// TIA Portal V20 export
// export: Created 2026-07-16T13:01:16.423654Z, ExportSetting WithDefaults, DisplayName Totally Integrated Automation Portal, DisplayVersion V20 Update 5, DisplayName TIA Portal Openness, DisplayVersion V20 Update 4, DisplayName TIA Portal Version Control Interface, DisplayVersion V20 Update 5, DisplayName SINAMICS Startdrive Advanced, DisplayVersion V20, DisplayName SINAMICS DCC, DisplayVersion V20, DisplayName SINAMICS Startdrive G130, G150, S120, S150, SINAMICS MV, G220, S200, S210, DisplayVersion V20, DisplayName SINAMICS Startdrive G110M, G120, G120C, G120D, G120P, G115D, DisplayVersion V20, DisplayName STEP 7 Professional, DisplayVersion V20 Update 5, DisplayName STEP 7 Safety, DisplayVersion V20 Update 2, DisplayName WinCC Basic/Comfort/Advanced, DisplayVersion V20 Update 5, DisplayName WinCC Unified, DisplayVersion V20 Update 5
VAR_GLOBAL   // PLC tag table "Default tag table"
   Tag_1 AT %I500.0 : Bool;
   Tag_2 AT %I500.1 : Bool;
   Tag_3 AT %I500.2 : Bool;
   Tag_4 AT %I500.3 : Bool;
   Tag_5 AT %I500.6 : Bool;
   Tag_6 AT %I500.7 : Bool;
   Tag_7 AT %I501.0 : Bool;
   Tag_8 AT %I501.1 : Bool;
   Tag_9 AT %I501.2 : Bool;
   Tag_10 AT %I501.3 : Bool;
   Tag_11 AT %I501.4 : Bool;
   Tag_12 AT %I501.5 : Bool;
   Tag_13 AT %I501.6 : Bool;
   Tag_14 AT %I501.7 : Bool;
   Tag_15 AT %I502.1 : Bool;
   Tag_16 AT %I502.2 : Bool;
   Tag_17 AT %I502.3 : Bool;
   Tag_18 AT %I502.4 : Bool;
   Tag_19 AT %I502.5 : Bool;
   Tag_20 AT %I502.6 : Bool;
   Tag_21 AT %I502.7 : Bool;
   Tag_22 AT %I503.0 : Bool;
   Tag_23 AT %I503.1 : Bool;
   Tag_24 AT %I503.2 : Bool;
   Tag_25 AT %I503.3 : Bool;
   Tag_26 AT %I503.4 : Bool;
   Tag_41 AT %IW508 : Word;
   Tag_42 AT %IW528 : Word;
   Tag_43 AT %IW532 : Word;
   Tag_44 AT %IW650 : Word;
   Tag_45 AT %IW64 : Word;
   Tag_46 AT %IW66 : Word;
   Tag_47 AT %IW68 : Word;
   Tag_48 AT %IW70 : Word;
   Tag_49 AT %IW72 : Word;
   Tag_50 AT %IW74 : Word;
   Tag_51 AT %IW76 : Word;
   Tag_52 AT %IW78 : Word;
   Tag_27 AT %Q500.0 : Bool;
   Tag_28 AT %Q500.1 : Bool;
   Tag_29 AT %Q500.2 : Bool;
   Tag_30 AT %Q500.4 : Bool;
   Tag_31 AT %Q500.5 : Bool;
   Tag_32 AT %Q501.0 : Bool;
   Tag_33 AT %Q501.1 : Bool;
   Tag_34 AT %Q501.2 : Bool;
   Tag_35 AT %Q501.3 : Bool;
   Tag_36 AT %Q501.4 : Bool;
   Tag_37 AT %Q501.5 : Bool;
   Tag_38 AT %Q502.0 : Bool;
   Tag_39 AT %Q502.1 : Bool;
   Tag_40 AT %Q502.2 : Bool;
   Tag_53 AT %QW64 : Word;
   Tag_54 AT %QW66 : Word;
   "Clock_0.5Hz" AT %M0.7 : Bool;
   AirStarWord0IN AT %IW80 : Word;
   AirStarWord2IN AT %IW82 : Word;
   AirStarWord0OUT AT %QW68 : Word;
   AirStarWord2OUT AT %QW70 : Word;
   FirstScan AT %M1.0 : Bool;
   AlwaysTrue AT %M1.2 : Bool;
   DI1_SYS_ControlHealthy AT %I0.0 : Bool;   // Safety/control circuit healthy
   DI2_SPR_1 AT %I0.1 : Bool;   // Spare (wired to -X3:1)
   DI3_SYS_CycleStart AT %I0.2 : Bool;   // Cycle start pushbutton (local/remote)
   DI4_SYS_CycleStop AT %I0.3 : Bool;   // Cycle stop pushbutton (NC)
   DI5_SHR_RunFwdFB AT %I0.4 : Bool;   // Shredder running forward feedback
   DI6_SHR_RunRevFB AT %I0.5 : Bool;   // Shredder running reverse feedback
   DI7_SYS_MotorFault AT %I0.6 : Bool;   // Motor fault (soft start fault relay)
   DI8_HPR_LevelHigh AT %I0.7 : Bool;   // Hopper high level sensor
   DI9_IFC_Running AT %I1.0 : Bool;   // Infeed conveyor running feedback
   DI10_DIS_Running AT %I1.1 : Bool;   // Discharge conveyor running feedback
   DI11_PSH_PowerPackRunning AT %I1.2 : Bool;   // Pusher power pack running feedback
   DI12_PSH_HomeLimit AT %I1.3 : Bool;   // Pusher parked/home position
   DI13_PSH_FullTravelLimit AT %I1.4 : Bool;   // Pusher fully extended position
   DI14_PSH_HighPressure AT %I1.5 : Bool;   // Pusher hydraulic high pressure switch
   DI15_SYS_DownstreamRunning AT %I2.0 : Bool;   // Downstream equipment running
   DI16_PSH_LocalRemote AT %I2.1 : Bool;   // Pusher operation local/remote selector
   DI17_SPR_2 AT %I2.2 : Bool;   // Spare (wired to terminal)
   DI18_SPR_3 AT %I2.3 : Bool;   // Spare (wired to terminal)
   DI19_SPR_4 AT %I2.4 : Bool;   // Spare (wired to terminal)
   DI20_SPR_5 AT %I2.5 : Bool;   // Spare (wired to terminal)
   DI21_SPR_6 AT %I2.6 : Bool;   // Spare (wired to terminal)
   DI22_SPR_7 AT %I2.7 : Bool;   // Spare (wired to terminal)
   DQ1_SHR_RunFwd AT %Q0.0 : Bool;   // Run shredder forward command
   DQ2_SHR_RunRev AT %Q0.1 : Bool;   // Run shredder reverse command
   DQ3_PSH_RunPowerPack AT %Q0.2 : Bool;   // Run pusher power pack command
   DQ4_IFC_Run AT %Q0.3 : Bool;   // Run infeed conveyor command
   DQ5_DIS_Run AT %Q0.4 : Bool;   // Run discharge conveyor command
   DQ6_PSH_Extend AT %Q0.5 : Bool;   // Pusher extend solenoid command
   DQ7_PSH_Retract AT %Q0.6 : Bool;   // Pusher retract solenoid command
   DQ8_SYS_InCycle AT %Q0.7 : Bool;   // Machine in-cycle status
   DQ9_SYS_EnableUpstream AT %Q1.0 : Bool;   // Enable upstream equipment (volt-free)
   DQ10_SYS_PreStartSounder AT %Q1.1 : Bool;   // Pre-start warning sounder/beacon
   DQ11_SHR_FaultReset AT %Q2.0 : Bool;   // Soft start motor fault reset
   DQ12_SPR_1 AT %Q2.1 : Bool;   // Spare (relay fitted)
   DQ13_SPR_2 AT %Q2.2 : Bool;   // Spare (relay fitted)
   DQ14_SPR_3 AT %Q2.3 : Bool;   // Spare (relay fitted)
   DQ15_SPR_4 AT %Q2.4 : Bool;   // Spare (relay fitted)
   DQ16_SPR_5 AT %Q2.5 : Bool;   // Spare (relay fitted)
   DQ17_SPR_6 AT %Q2.6 : Bool;   // Spare (wired to -X13:6)
   DQ18_SPR_7 AT %Q2.7 : Bool;   // Spare (wired to -X13:7)
END_VAR
